// TIA Portal project "PALLETA_GEP_VEZERLES-1500_V15" (V15)

(* hardware
DEVICE "S71500/ET200MP-Station_1"  S7-1500 station
   slot 0: "Profilschiene_0"  6ES7 590-1***0-0AA0
   slot 1: "PLC_1"  CPU 1511-1 PN  6ES7 511-1AK00-0AB0  V1.8
   slot 2: "AI 8xU/I/RTD/TC ST_1"  AI 8xU/I/RTD/TC ST  6ES7 531-7KF00-0AB0  V2.0
   slot 3: "AI 8xU/I/RTD/TC ST_2"  AI 8xU/I/RTD/TC ST  6ES7 531-7KF00-0AB0  V2.0
   slot 4: "AI 8xU/I/RTD/TC ST_3"  AI 8xU/I/RTD/TC ST  6ES7 531-7KF00-0AB0  V2.0
   slot 5: "AI 8xU/I/RTD/TC ST_4"  AI 8xU/I/RTD/TC ST  6ES7 531-7KF00-0AB0  V2.0
   slot 6: "DI 16x24VDC BA_1"  DI 16x24VDC BA  6ES7 521-1BH10-0AA0  V1.0
*)

// ===== PLC "PLC_1"  CPU 1511-1 PN =====

VAR_GLOBAL   // PLC tag table "Standard-Variablentabelle"
   "PALLET_AT_ENTRY" AT %I0.0 : Bool;
   "PALLET_AT_EXIT" AT %I0.1 : Bool;
   "PALLET_LOADED" AT %I0.2 : Bool;
   "BOX_AT_ENTRY" AT %I0.3 : Bool;
   "PUSHER_LIMIT" AT %I0.4 : Bool;
   "PLATE_LIMIT" AT %I0.5 : Bool;
   "CLAMPED" AT %I0.6 : Bool;
   "ELEVATOR_MOVING" AT %I0.7 : Bool;
   "START" AT %I1.0 : Bool;
   "RESET" AT %I1.1 : Bool;
   "STOP" AT %I1.2 : Bool;
   "EM_STOP" AT %I1.3 : Bool;
   "AUTO" AT %I1.4 : Bool;
   "PALLET_FEEDER" AT %Q0.0 : Bool;
   "LOAD_PALLET" AT %Q0.1 : Bool;
   "EXIT_CONVEYOR" AT %Q0.2 : Bool;
   "MOVE_TO_LIMIT" AT %Q0.3 : Bool;
   "ELEVATOR_UP" AT %Q0.4 : Bool;
   "ELEVATOR_DOWN" AT %Q0.5 : Bool;
   "TURN" AT %Q0.7 : Bool;
   "PUSH" AT %Q1.0 : Bool;
   "LOAD_BELT" AT %Q1.1 : Bool;
   "CLAMP" AT %Q1.2 : Bool;
   "WARNING_LIGHT" AT %Q1.4 : Bool;
   "RESET_LIGHT" AT %Q1.5 : Bool;
   "STOP_LIGHT" AT %Q1.6 : Bool;
   "BOX_FEEDER" AT %Q0.6 : Bool;
   "OPEN_PLATE" AT %Q1.3 : Bool;
END_VAR

DATA_BLOCK "mainProgram_DB"   // DB1
{ S7_Optimized_Access := 'TRUE' }
VERSION : 0.1
// stored: InstanceOfName mainProgram
"mainProgram"
BEGIN
END_DATA_BLOCK

// folder: System blocks/Program resources

DATA_BLOCK "IEC_Timer_0_DB"   // DB7
{ S7_Optimized_Access := 'TRUE' }
AUTHOR : Simatic
FAMILY : IEC
NAME : IEC_TMR
VERSION : 1.0
// stored: InstanceOfName IEC_TIMER
"IEC_TIMER"
BEGIN
END_DATA_BLOCK

DATA_BLOCK "IEC_Timer_0_DB_1"   // DB9
{ S7_Optimized_Access := 'TRUE' }
AUTHOR : Simatic
FAMILY : IEC
NAME : IEC_TMR
VERSION : 1.0
// stored: InstanceOfName IEC_TIMER
"IEC_TIMER"
BEGIN
END_DATA_BLOCK

DATA_BLOCK "IEC_Timer_0_DB_2"   // DB11
{ S7_Optimized_Access := 'TRUE' }
AUTHOR : Simatic
FAMILY : IEC
NAME : IEC_TMR
VERSION : 1.0
// stored: InstanceOfName IEC_TIMER
"IEC_TIMER"
BEGIN
END_DATA_BLOCK

DATA_BLOCK "IEC_Timer_0_DB_3"   // DB13
{ S7_Optimized_Access := 'TRUE' }
AUTHOR : Simatic
FAMILY : IEC
NAME : IEC_TMR
VERSION : 1.0
// stored: InstanceOfName IEC_TIMER
"IEC_TIMER"
BEGIN
END_DATA_BLOCK

// folder: (top level)

FUNCTION_BLOCK "mainProgram"   // FB1, SCL
{ S7_Optimized_Access := 'TRUE' }
VERSION : 0.1
   VAR_INPUT
      palletAtEntry : Bool;
      palletAtExit : Bool;
      palletLoaded : Bool;
      boxAtEntry : Bool;
      pusherLinit : Bool;
      plateeLimit : Bool;
      clamped : Bool;
      elevatorMoving : Bool;
      start : Bool;
      reset : Bool;
      stop : Bool;
      emStop : Bool;
      auto : Bool;
   END_VAR
   VAR_OUTPUT
      palletFeeder : Bool;
      loadPallet : Bool;
      exitConveyor : Bool;
      moveToLinit : Bool;
      elevatorUp : Bool;
      elevatorDown : Bool;
      boxFeeder : Bool;
      turn : Bool;
      push : Bool;
      loadBelt : Bool;
      clamp : Bool;
      openPlate : Bool;
      warningLight : Bool;
      startLight : Bool;
      resetLight : Bool;
      stopLight : Bool;
   END_VAR
   VAR
      currentState : Int;
      boxInPalletCounter : Int;
      boxCounter : Int;
      maxBoxes : Int := 1;
      maxBoxInPallet : Int;
      "counter" : Int;
      palletWaitTime : Time := T#3s;
      risingEgdeDedect : Bool;
      fallingEgdeDedect : Bool;
      onDelayTimerCheck : Bool;
      rotateBoxes : Bool;
      firstPalletArrived : Bool;
      firstBoxesArrived : Bool;
      firstRowOfPalletCompleted : Bool;
      processFinished : Bool;
      "timer" : Time;
   END_VAR
   VAR CONSTANT
      PALLETE_UP_IMPULSE : Int := 14;
      PALLET_WAIT_TIME : Time := T#3150ms;
      MAX_BOX_IN_PALLETE : Int := 4;
      MAX_BOX_COUNT : Int := 2;
      STATE_INIT : Int;
      STATE_START_BOX_FEED : Int := 1;
      STATE_COUNT_BOXES : Int := 2;
      STATE_STOP_BOX_FEED : Int := 3;
      STATE_START_PUSH_BOXES : Int := 4;
      STATE_STOP_PUSH_BOXES : Int := 5;
      STATE_MOVE_PALLET_TO_ELEVATOR : Int := 6;
      STATE_STOP_PALLET_AT_ELEVATOR : Int := 7;
      STATE_MOVE_PALLET_UP_WITH_ELEVATOR : Int := 8;
      STATE_OPEN_PALLET_WINDOW : Int := 9;
      STATE_MOVE_ELEVATOR_BY_ONE_LEVEL : Int := 10;
      STATE_MOVE_PALLETE_DOWN : Int := 11;
      STATE_MOVE_PALLET_TO_EXIT : Int := 12;
   END_VAR
BEGIN
     CASE #currentState OF
       #STATE_INIT:
           "R_TRIG_DB"(CLK := #start,
                       Q => #risingEgdeDedect);

           IF #risingEgdeDedect THEN
               #currentState := #STATE_START_BOX_FEED;
               #maxBoxInPallet := #MAX_BOX_IN_PALLETE;
           END_IF;

       #STATE_START_BOX_FEED:
           #boxFeeder := TRUE;
           #loadBelt := TRUE;

           IF #rotateBoxes THEN
               #turn := TRUE;
           ELSE
               #turn := FALSE;
           END_IF;

           IF #firstBoxesArrived AND NOT #rotateBoxes THEN
               #maxBoxes := #MAX_BOX_COUNT;
               #maxBoxInPallet := #MAX_BOX_IN_PALLETE;
           END_IF;

           IF #firstBoxesArrived AND NOT #rotateBoxes AND #processFinished THEN
               #maxBoxes := #MAX_BOX_COUNT;
               #maxBoxInPallet := #MAX_BOX_IN_PALLETE - 1;
           END_IF;

           IF #firstBoxesArrived AND #rotateBoxes THEN
               #warningLight := TRUE;
               #maxBoxes := #MAX_BOX_COUNT + 1;
               #maxBoxInPallet := #MAX_BOX_IN_PALLETE - 2;
           END_IF;

           IF #firstPalletArrived THEN
               #palletWaitTime := #PALLET_WAIT_TIME;
           END_IF;

           #currentState := #STATE_COUNT_BOXES;

       #STATE_COUNT_BOXES:
           "F_TRIG_DB"(CLK := #boxAtEntry,
                       Q => #fallingEgdeDedect);

           IF #fallingEgdeDedect THEN
               #fallingEgdeDedect := TRUE;
               #boxCounter += 1;
           END_IF;

           IF #boxCounter = #maxBoxes THEN
               #currentState := #STATE_STOP_BOX_FEED;
               #boxCounter := 0;
           END_IF;

       #STATE_STOP_BOX_FEED:
           #boxFeeder := FALSE;
           #loadBelt := FALSE;
           #currentState := #STATE_START_PUSH_BOXES;

       #STATE_START_PUSH_BOXES:
           #push := TRUE;

           "R_TRIG_DB_1"(CLK := #pusherLinit,
                         Q => #risingEgdeDedect);

           IF #risingEgdeDedect THEN
               #risingEgdeDedect := FALSE;
               #boxInPalletCounter += 1;
               #currentState := #STATE_STOP_PUSH_BOXES;
           END_IF; 

       #STATE_STOP_PUSH_BOXES:
           #push := FALSE;

           "R_TRIG_DB_2"(CLK:=#pusherLinit,
                         Q=>#risingEgdeDedect);

           IF #risingEgdeDedect AND #boxInPalletCounter < #maxBoxInPallet THEN
               #currentState := #STATE_START_BOX_FEED;
               #risingEgdeDedect := FALSE;
               #firstBoxesArrived := TRUE;
           END_IF;

           IF #risingEgdeDedect AND #boxInPalletCounter = #maxBoxInPallet THEN
               IF #rotateBoxes THEN
                   #currentState := #STATE_OPEN_PALLET_WINDOW;
                   #boxInPalletCounter := 0;
                   #risingEgdeDedect := FALSE;
                   #firstBoxesArrived := TRUE;
               ELSE
                   #currentState := #STATE_MOVE_PALLET_TO_ELEVATOR;
                   #boxInPalletCounter := 0;
                   #risingEgdeDedect := FALSE;
                   #firstBoxesArrived := TRUE;
               END_IF;
           END_IF;

       #STATE_MOVE_PALLET_TO_ELEVATOR:
           #palletFeeder := TRUE;
           #loadPallet := TRUE;

           "F_TRIG_DB_1"(CLK:=#palletAtEntry,
                         Q=>#fallingEgdeDedect);

           IF #firstPalletArrived THEN
               #currentState := #STATE_STOP_PALLET_AT_ELEVATOR;
           END_IF;

           IF #fallingEgdeDedect AND NOT #firstPalletArrived THEN
               #fallingEgdeDedect := FALSE;
               #currentState := #STATE_STOP_PALLET_AT_ELEVATOR;
               #firstPalletArrived := TRUE;
           END_IF;

       #STATE_STOP_PALLET_AT_ELEVATOR:
           "IEC_Timer_0_DB".TON(IN := TRUE,
                                PT := #palletWaitTime,
                                Q => #onDelayTimerCheck,
                                ET => #timer);

           IF #onDelayTimerCheck THEN
               #palletFeeder := FALSE;
               #loadPallet := FALSE;
               #currentState := #STATE_MOVE_PALLET_UP_WITH_ELEVATOR;
               "IEC_Timer_0_DB".TON(IN:=FALSE, PT:=T#1s);
           END_IF;

       #STATE_MOVE_PALLET_UP_WITH_ELEVATOR:
           #moveToLinit := TRUE;
           #elevatorUp := TRUE;

           "F_TRIG_DB_2"(CLK:=#elevatorMoving,
                         Q=>#fallingEgdeDedect);

           IF #fallingEgdeDedect THEN
               #moveToLinit := FALSE;
               #elevatorUp := FALSE;
               #currentState := #STATE_OPEN_PALLET_WINDOW;
           END_IF;

       #STATE_OPEN_PALLET_WINDOW:
           #openPlate := TRUE;

           "IEC_Timer_0_DB_1".TON(IN:=TRUE,
                                  PT:=T#8s,
                                  Q=>#onDelayTimerCheck,
                                  ET=>#timer);

           IF #onDelayTimerCheck THEN
               "IEC_Timer_0_DB_1".TON(IN := FALSE,
                                      PT := T#5s);

               #currentState := #STATE_MOVE_ELEVATOR_BY_ONE_LEVEL;
           END_IF;

       #STATE_MOVE_ELEVATOR_BY_ONE_LEVEL:
           "IEC_Timer_0_DB_3".TP(IN:=TRUE,
                                 PT:=T#500ms,
                                 Q=>#elevatorDown,
                                 ET=>#timer);

           "F_TRIG_DB_5"(CLK:=#elevatorMoving,
                         Q=>#fallingEgdeDedect);

           IF #fallingEgdeDedect THEN
               #openPlate := FALSE;
               "IEC_Timer_0_DB_3".TP(IN := FALSE,
                                     PT := T#500ms);

               IF #rotateBoxes THEN
                   #currentState := #STATE_MOVE_PALLETE_DOWN;
               ELSE
                   #currentState := #STATE_START_BOX_FEED;
                   #rotateBoxes := TRUE;
               END_IF;

           END_IF;

       #STATE_MOVE_PALLETE_DOWN:
           #moveToLinit := TRUE;
           #elevatorDown := TRUE;
           #openPlate := FALSE;

           "F_TRIG_DB_3"(CLK:=#elevatorMoving,
                         Q=>#fallingEgdeDedect);

           IF #fallingEgdeDedect THEN
               #moveToLinit := FALSE;
               #elevatorDown := FALSE;
               #currentState := #STATE_MOVE_PALLET_TO_EXIT;
           END_IF;

       #STATE_MOVE_PALLET_TO_EXIT:
           #exitConveyor := TRUE;
           #loadPallet := TRUE;

           "IEC_Timer_0_DB_2".TON(IN:=TRUE,
                                  PT:=T#10s,
                                  Q=>#onDelayTimerCheck,
                                  ET=>#timer);

           IF #onDelayTimerCheck THEN
               #exitConveyor := FALSE;
               #loadPallet := FALSE;
               "IEC_Timer_0_DB_2".TON(IN := FALSE,
                                      PT := T#10s);
               #currentState := #STATE_START_BOX_FEED;
               #rotateBoxes := FALSE;
               #boxCounter := 0;
               #boxInPalletCounter := 0;
               #processFinished := TRUE;
           END_IF;
   END_CASE;
END_FUNCTION_BLOCK

FUNCTION "MHJ-PLC-Lab-Function-S71500" : Void   // FC9000, SCL
{ S7_Optimized_Access := 'TRUE' }
VERSION : 0.1
   VAR_TEMP
      Value : Byte;
      ForCounter : Int;
   END_VAR
   VAR CONSTANT
      Value_01_DW : DWord := 16#1223_5486;
      Value_02_DW : DWord := 16#A6C9_D1F5;
   END_VAR
BEGIN

   #Value:=PEEK(area := 16#82,
        dbNumber := 0,
        byteOffset := 511);
   #Value := #Value + 1;

   POKE(area := 16#82,
        dbNumber := 0,
        byteOffset := 511,
        value := #Value);

   POKE(area := 16#82,
        dbNumber := 0,
        byteOffset := 1016,
        value := #Value_01_DW);
   POKE(area := 16#82,
        dbNumber := 0,
        byteOffset := 1020,
        value := #Value_02_DW);

   FOR #ForCounter := 0 TO 63 DO
       #Value:=PEEK(area := 16#1,
            dbNumber := 0,
            byteOffset := #ForCounter);
       POKE(area := 16#81,
            dbNumber := 0,
            byteOffset := #ForCounter,
            value := #Value);
   END_FOR;
   #Value := PEEK(area := 16#1,
                  dbNumber := 0,
                  byteOffset := 512);
   POKE(area := 16#82,
        dbNumber := 0,
        byteOffset := 512,
        value := #Value);
END_FUNCTION

ORGANIZATION_BLOCK "Main"   // OB1, FBD, ProgramCycle
TITLE = "Main Program Sweep (Cycle)"
{ S7_Optimized_Access := 'TRUE' }
VERSION : 0.1
   VAR_INPUT
      Initial_Call : Bool;   // Initial call of this OB
      Remanence : Bool;   // =True, if remanent data are available
   END_VAR
BEGIN

REGION Network 1
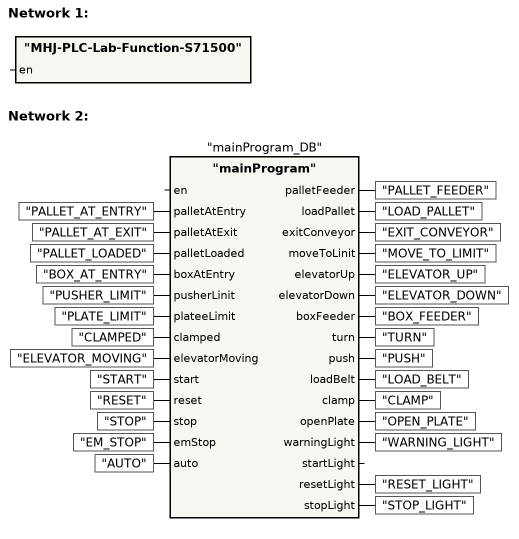
   "MHJ-PLC-Lab-Function-S71500"();
END_REGION

REGION Network 2
   "mainProgram_DB"(palletAtEntry := "PALLET_AT_ENTRY",   // "mainProgram"
                    palletAtExit := "PALLET_AT_EXIT",
                    palletLoaded := "PALLET_LOADED",
                    boxAtEntry := "BOX_AT_ENTRY",
                    pusherLinit := "PUSHER_LIMIT",
                    plateeLimit := "PLATE_LIMIT",
                    clamped := "CLAMPED",
                    elevatorMoving := "ELEVATOR_MOVING",
                    start := "START",
                    reset := "RESET",
                    stop := "STOP",
                    emStop := "EM_STOP",
                    auto := "AUTO",
                    palletFeeder => "PALLET_FEEDER",
                    loadPallet => "LOAD_PALLET",
                    exitConveyor => "EXIT_CONVEYOR",
                    moveToLinit => "MOVE_TO_LIMIT",
                    elevatorUp => "ELEVATOR_UP",
                    elevatorDown => "ELEVATOR_DOWN",
                    boxFeeder => "BOX_FEEDER",
                    turn => "TURN",
                    push => "PUSH",
                    loadBelt => "LOAD_BELT",
                    clamp => "CLAMP",
                    openPlate => "OPEN_PLATE",
                    warningLight => "WARNING_LIGHT",
                    resetLight => "RESET_LIGHT",
                    stopLight => "STOP_LIGHT");
END_REGION
END_ORGANIZATION_BLOCK